// TIA Portal V20 export
FUNCTION_BLOCK "sleepModeManager"   // FB80, LAD
// stored: Access Published, MemoryReserve 100, SetENOAutomatically false
   VAR_INPUT
      mode : "LER_typeSleepMode";
      configuration : "LER_typeSleepModeParameter";
      Reset : Bool;
   END_VAR
   VAR_OUTPUT
      CurrentMode : "LER_typeSleepMode";
      Output : "LER_typeSleep";
      sleepTime : Time;
      deepSleepTime : Time;
   END_VAR
   VAR
      instTimer_ton : Array[0..2] of TON_TIME;
   END_VAR
   VAR CONSTANT
      TRUE : Bool := TRUE;
      FALSE : Bool := FALSE;
   END_VAR
   VAR_TEMP   // added for the SCL form of the ladder/FBD networks
      _w1 : Bool;
      _w2 : Bool;
      _w3 : Bool;
      _w4 : Bool;
   END_VAR
BEGIN

REGION Network 1: State
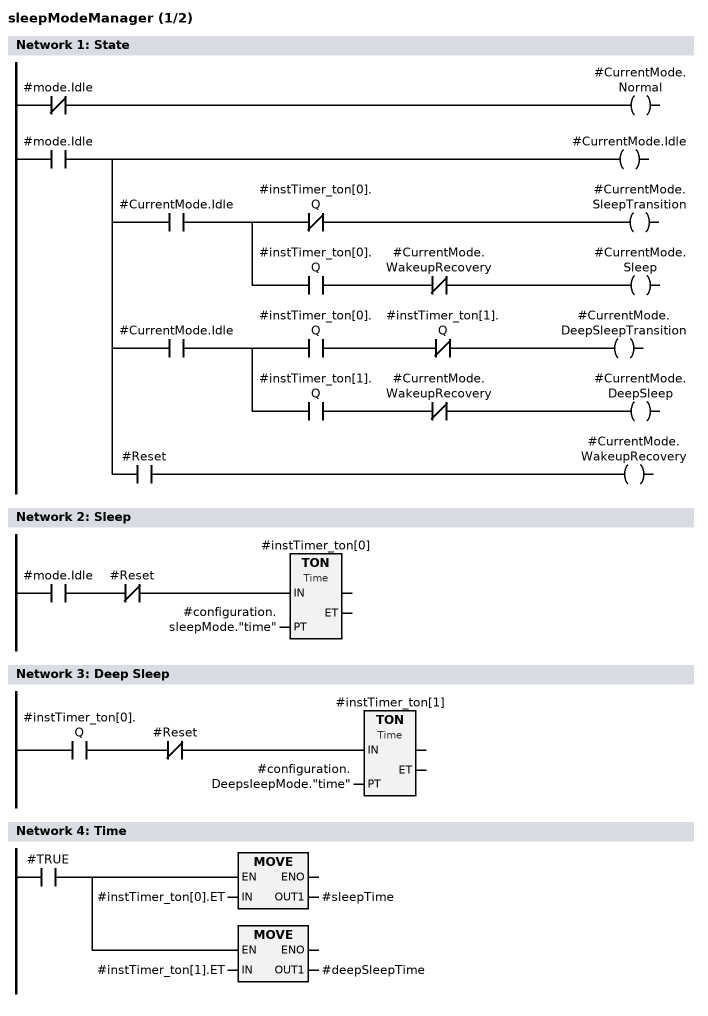
   RUNG wire#powerrail
      I_Contact( #mode.Idle )
      Coil( #CurrentMode.Normal )
   END_RUNG
   RUNG wire#powerrail
      Contact( #mode.Idle )
      wire#w1
      Coil( #CurrentMode.Idle )
   END_RUNG
   RUNG wire#w1
      Contact( #CurrentMode.Idle )
      wire#w2
      I_Contact( #instTimer_ton[0].Q )
      Coil( #CurrentMode.SleepTransition )
   END_RUNG
   RUNG wire#w2
      Contact( #instTimer_ton[0].Q )
      I_Contact( #CurrentMode.WakeupRecovery )
      Coil( #CurrentMode.Sleep )
   END_RUNG
   RUNG wire#w1
      Contact( #CurrentMode.Idle )
      wire#w3
      Contact( #instTimer_ton[0].Q )
      I_Contact( #instTimer_ton[1].Q )
      Coil( #CurrentMode.DeepSleepTransition )
   END_RUNG
   RUNG wire#w3
      Contact( #instTimer_ton[1].Q )
      I_Contact( #CurrentMode.WakeupRecovery )
      Coil( #CurrentMode.DeepSleep )
   END_RUNG
   RUNG wire#w1
      Contact( #Reset )
      Coil( #CurrentMode.WakeupRecovery )
   END_RUNG
   // the same network as SCL:
   #CurrentMode.Normal := NOT #mode.Idle;
   #CurrentMode.Idle := #mode.Idle;
   #_w1 := #mode.Idle AND #CurrentMode.Idle;
   #CurrentMode.SleepTransition := #_w1 AND NOT #instTimer_ton[0].Q;
   #CurrentMode.Sleep := #_w1 AND #instTimer_ton[0].Q AND NOT #CurrentMode.WakeupRecovery;
   #_w2 := #mode.Idle AND #CurrentMode.Idle;
   #CurrentMode.DeepSleepTransition := #_w2 AND #instTimer_ton[0].Q AND NOT #instTimer_ton[1].Q;
   #CurrentMode.DeepSleep := #_w2 AND #instTimer_ton[1].Q AND NOT #CurrentMode.WakeupRecovery;
   #CurrentMode.WakeupRecovery := #mode.Idle AND #Reset;
END_REGION

REGION Network 2: Sleep
   RUNG wire#powerrail
      Contact( #mode.Idle )
      I_Contact( #Reset )
      { S7_Templates := "time_type := Time" } #instTimer_ton[0].TON(pt := #configuration.sleepMode."time", et =>)
   END_RUNG
   // the same network as SCL:
   #instTimer_ton[0].TON(IN := #mode.Idle AND NOT #Reset, PT := #configuration.sleepMode."time");
END_REGION

REGION Network 3: Deep Sleep
   RUNG wire#powerrail
      Contact( #instTimer_ton[0].Q )
      I_Contact( #Reset )
      { S7_Templates := "time_type := Time" } #instTimer_ton[1].TON(pt := #configuration.DeepsleepMode."time", et =>)
   END_RUNG
   // the same network as SCL:
   #instTimer_ton[1].TON(IN := #instTimer_ton[0].Q AND NOT #Reset, PT := #configuration.DeepsleepMode."time");
END_REGION

REGION Network 4: Time
   RUNG wire#powerrail
      Contact( #TRUE )
      wire#w1
      Move(in := #instTimer_ton[0].ET, out1 => #sleepTime)
   END_RUNG
   RUNG wire#w1
      Move(in := #instTimer_ton[1].ET, out1 => #deepSleepTime)
   END_RUNG
   // the same network as SCL:
   IF #TRUE THEN
       #sleepTime := #instTimer_ton[0].ET;
       #deepSleepTime := #instTimer_ton[1].ET;
   END_IF;
END_REGION

REGION Network 5: Sleep Output
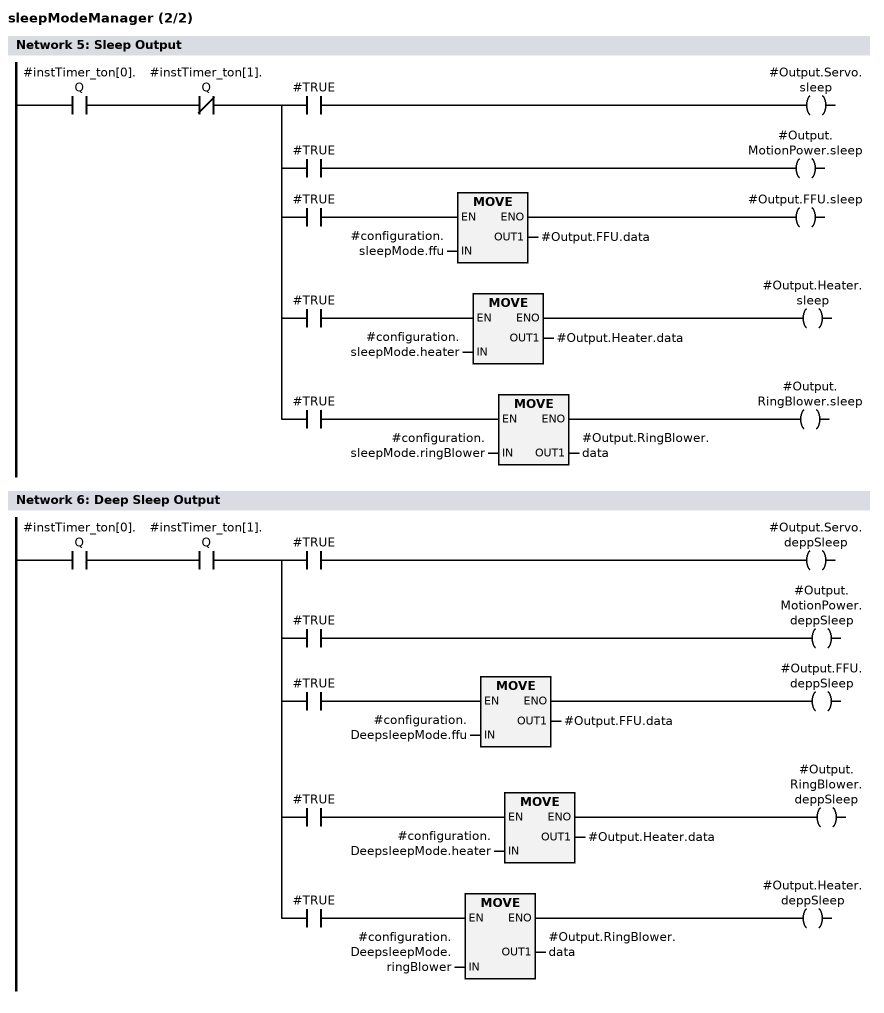
   RUNG wire#powerrail
      Contact( #instTimer_ton[0].Q )
      I_Contact( #instTimer_ton[1].Q )
      wire#w1
      Contact( #TRUE )
      Coil( #Output.Servo.sleep )
   END_RUNG
   RUNG wire#w1
      Contact( #TRUE )
      Coil( #Output.MotionPower.sleep )
   END_RUNG
   RUNG wire#w1
      Contact( #TRUE )
      Move(in := #configuration.sleepMode.ffu, out1 => #Output.FFU.data)
      Coil( #Output.FFU.sleep )
   END_RUNG
   RUNG wire#w1
      Contact( #TRUE )
      Move(in := #configuration.sleepMode.heater, out1 => #Output.Heater.data)
      Coil( #Output.Heater.sleep )
   END_RUNG
   RUNG wire#w1
      Contact( #TRUE )
      Move(in := #configuration.sleepMode.ringBlower, out1 => #Output.RingBlower.data)
      Coil( #Output.RingBlower.sleep )
   END_RUNG
   // the same network as SCL:
   #_w1 := #instTimer_ton[0].Q AND NOT #instTimer_ton[1].Q;
   #Output.Servo.sleep := #_w1 AND #TRUE;
   #Output.MotionPower.sleep := #_w1 AND #TRUE;
   #_w2 := #_w1 AND #TRUE;
   IF #_w2 THEN #Output.FFU.data := #configuration.sleepMode.ffu; END_IF;
   #Output.FFU.sleep := #_w2;
   #_w3 := #_w1 AND #TRUE;
   IF #_w3 THEN #Output.Heater.data := #configuration.sleepMode.heater; END_IF;
   #Output.Heater.sleep := #_w3;
   #_w4 := #_w1 AND #TRUE;
   IF #_w4 THEN #Output.RingBlower.data := #configuration.sleepMode.ringBlower; END_IF;
   #Output.RingBlower.sleep := #_w4;
END_REGION

REGION Network 6: Deep Sleep Output
   RUNG wire#powerrail
      Contact( #instTimer_ton[0].Q )
      Contact( #instTimer_ton[1].Q )
      wire#w1
      Contact( #TRUE )
      Coil( #Output.Servo.deppSleep )
   END_RUNG
   RUNG wire#w1
      Contact( #TRUE )
      Coil( #Output.MotionPower.deppSleep )
   END_RUNG
   RUNG wire#w1
      Contact( #TRUE )
      Move(in := #configuration.DeepsleepMode.ffu, out1 => #Output.FFU.data)
      Coil( #Output.FFU.deppSleep )
   END_RUNG
   RUNG wire#w1
      Contact( #TRUE )
      Move(in := #configuration.DeepsleepMode.heater, out1 => #Output.Heater.data)
      Coil( #Output.RingBlower.deppSleep )
   END_RUNG
   RUNG wire#w1
      Contact( #TRUE )
      Move(in := #configuration.DeepsleepMode.ringBlower, out1 => #Output.RingBlower.data)
      Coil( #Output.Heater.deppSleep )
   END_RUNG
   // the same network as SCL:
   #_w1 := #instTimer_ton[0].Q AND #instTimer_ton[1].Q;
   #Output.Servo.deppSleep := #_w1 AND #TRUE;
   #Output.MotionPower.deppSleep := #_w1 AND #TRUE;
   #_w2 := #_w1 AND #TRUE;
   IF #_w2 THEN #Output.FFU.data := #configuration.DeepsleepMode.ffu; END_IF;
   #Output.FFU.deppSleep := #_w2;
   #_w3 := #_w1 AND #TRUE;
   IF #_w3 THEN #Output.Heater.data := #configuration.DeepsleepMode.heater; END_IF;
   #Output.RingBlower.deppSleep := #_w3;
   #_w4 := #_w1 AND #TRUE;
   IF #_w4 THEN #Output.RingBlower.data := #configuration.DeepsleepMode.ringBlower; END_IF;
   #Output.Heater.deppSleep := #_w4;
END_REGION
END_FUNCTION_BLOCK
